TYPE ST_P_START_ASSY :
STRUCT
	Barcode:				INT;
END_STRUCT
END_TYPE

(* stored: Version 1.1.0.1, ProductVersion 3.1.4024.10
   DUT ST_P_START_ASSY: Id {82b0ddcd-5a86-4b4e-9f7a-edf6b43808ba} *)
